FUNCTION_BLOCK OrchestratorExample (* Template for a simple Basic Function Block Type *)
  (* Standard: 61499-2 *)
  (* Version 1.0, 2019-11-08, dorofeev *)
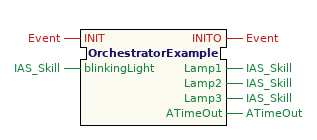
  EVENT_INPUT
    INIT; (* Initialization Request *)
  END_EVENT
  EVENT_OUTPUT
    INITO; (* Initialization Confirm *)
  END_EVENT
  SOCKETS
    blinkingLight : IAS_Skill;
  END_SOCKETS
  PLUGS
    Lamp1 : IAS_Skill;
    Lamp2 : IAS_Skill;
    Lamp3 : IAS_Skill;
    ATimeOut : ATimeOut;
  END_PLUGS
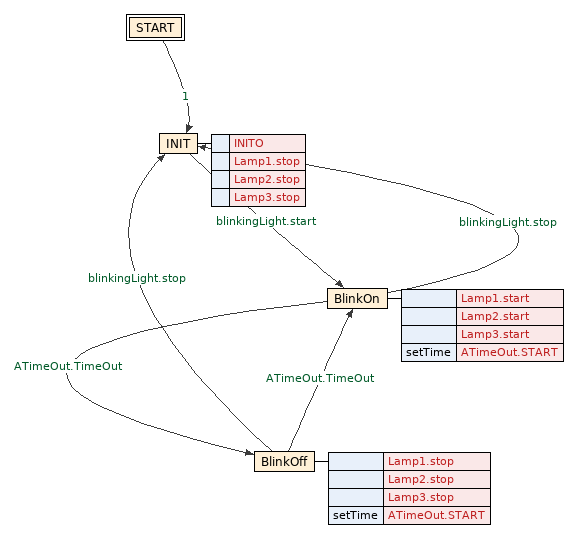
  EC_STATES
    START; (* Initial State *)
    BlinkOn : -> Lamp1.start, -> Lamp2.start, -> Lamp3.start, setTime -> ATimeOut.START;
    BlinkOff : -> Lamp1.stop, -> Lamp2.stop, -> Lamp3.stop, setTime -> ATimeOut.START;
    INIT : -> INITO, -> Lamp1.stop, -> Lamp2.stop, -> Lamp3.stop;
  END_STATES
  EC_TRANSITIONS
    BlinkOn TO BlinkOff := ATimeOut.TimeOut;
    BlinkOff TO BlinkOn := ATimeOut.TimeOut;
    INIT TO BlinkOn := blinkingLight.start;
    BlinkOff TO INIT := blinkingLight.stop;
    START TO INIT := 1;
    BlinkOn TO INIT := blinkingLight.stop;
  END_TRANSITIONS
  ALGORITHM setTime IN ST: (* new algorithm *)
ATimeOut.DT := T#5s;
  END_ALGORITHM
END_FUNCTION_BLOCK
